PROGRAM Balanza_Semilla
VAR
	// grueso carga balanza
	TR_S_V2: Equipo_Valvula_5_2; //Válvula de corte grosso
	// fino carga balanza
	TR_S_V3: Equipo_Valvula_5_2;
	// descarga balanza
	TR_S_V4: Equipo_Valvula_5_2;
	//
	TR_S_V2_CmdAuto:BOOL;	//Válvula de corte grosso
	TR_S_V3_CmdAuto:BOOL;	//Válvula de corte fino
	TR_S_V4_CmdAuto:BOOL;	//Válvula de descarga
	// Balanza de pesaje de semilla
	TR_S_WT1: Balanza;
	//
	Hab_cargarSemilla	:BOOL;
	Cargar_Balanza		:BOOL;
	TolerInf_pesoSemilla:REAL;	//Tolerância inferior da carga da balança
	TolerSup_pesoSemilla:REAL;	//Tolerância superior da balança
	Balanza_cargadaOk	:BOOL;
	Hab_descargarSemilla:BOOL;
	Descargar_Balanza	:BOOL;
	PesoSemilla_paraDosificar:REAL;
	Espera_pesasArriba:TON;
	Espera_Estable:TON;
	Espera_DescAbierta:TON;
	
	// tiempo de carga/descarga de balanza semilla excesivo
	Alr_demoraCarga: TON;
	Alr_demoraDescarga:TON;
	
	TriggerTomarPeso :BOOL;
	
	//provisorios
	bHS :BOOL;
	dintHS	:DINT:=3;
	Hx :BOOL;
	IniCal:BOOL;
	
	iStep :INT;
	Espera_pesas :TON;
	
	AuxHugo :BOOL;
	Procesando: BOOL;
	Tabla_FIFO_Peso: Tabla_FIFO;
	Balanza_vacia: BOOL;
	FinCarga: BOOL;
	TmrGruesoOk: TON;
	TBalanzaVacia: TON;
	PolvosOk: BOOL;
	// Timer para aparecer a popup de peso fora de tolerância
	TON_PesoForaTolerancia: TON;
	TON_DemoraCarga: TON;
	// Se a caixa superior estiver sem nível de sementes, permite que a semente remanescente seja carregada na balança
	EsvaziarCaixa: BOOL;
	qtdBateladas	:UDINT;	//Quantidade de bateladas feitas
END_VAR
VAR // added by the converter: edge detectors and wires of the graphical bodies
    _rt1, _rt2, _rt3, _rt4, _rt5, _rt6 : R_TRIG;
    _w1, _w2, _w3, _w4, _w5, _w6, _w7, _w8, _w9, _w10, _w11, _w12, _w13, _w14, _w15 : BOOL;
    _ft1 : F_TRIG;
END_VAR

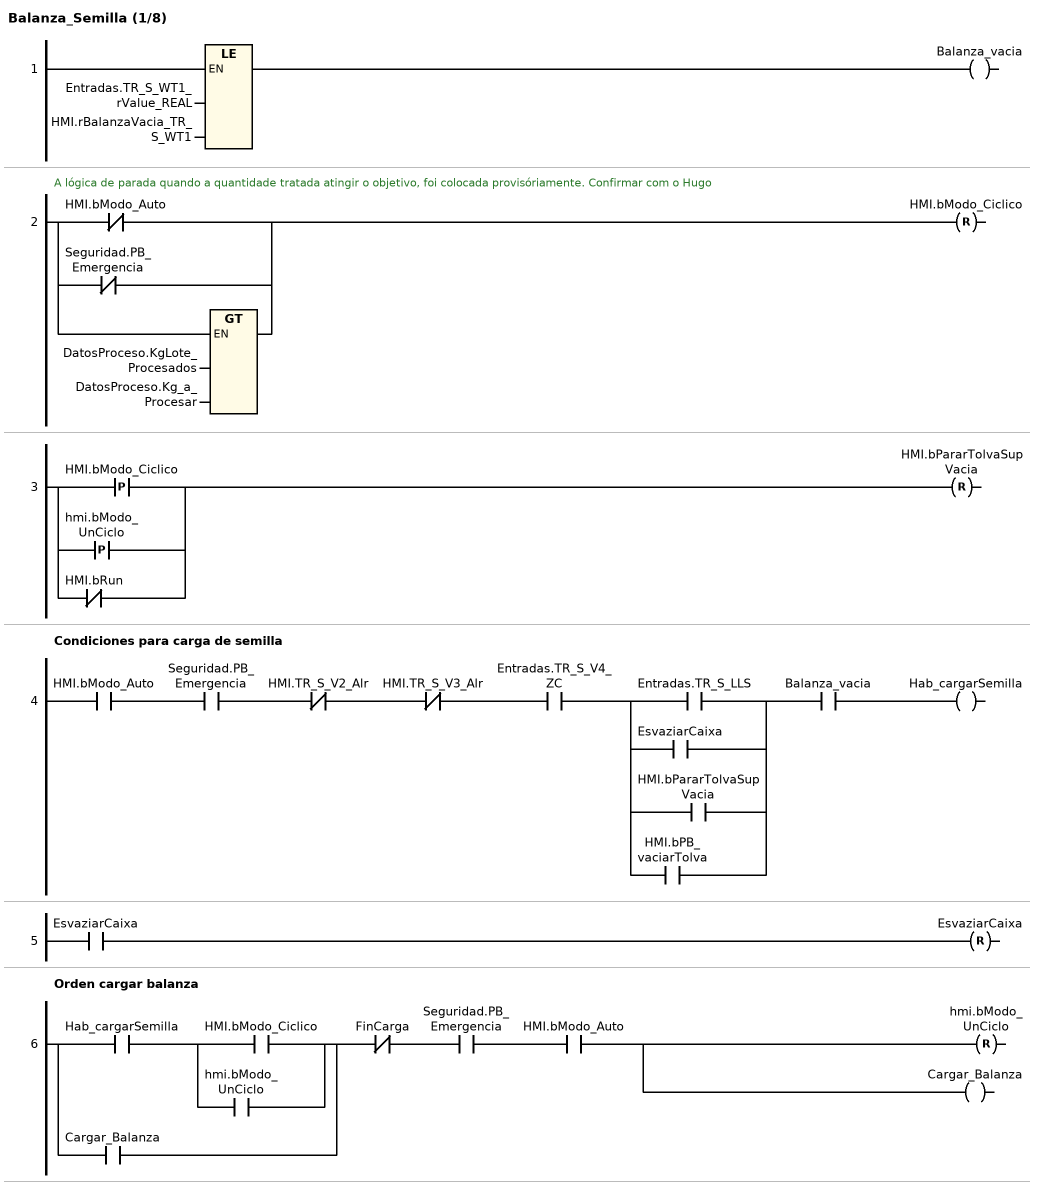
// NETWORK 1
Balanza_vacia := Entradas.TR_S_WT1_rValue_REAL <= HMI.rBalanzaVacia_TR_S_WT1;

// NETWORK 2
// A lógica de parada quando a quantidade tratada atingir o objetivo, foi colocada provisóriamente. Confirmar com o Hugo
HMI.bModo_Ciclico R= NOT HMI.bModo_Auto OR NOT Seguridad.PB_Emergencia OR DatosProceso.KgLote_Procesados > DatosProceso.Kg_a_Procesar;

// NETWORK 3
_rt1(CLK := HMI.bModo_Ciclico);
_rt2(CLK := hmi.bModo_UnCiclo);
HMI.bPararTolvaSupVacia R= _rt1.Q OR _rt2.Q OR NOT HMI.bRun;

// NETWORK 4: Condiciones para carga de semilla
Hab_cargarSemilla := HMI.bModo_Auto AND Seguridad.PB_Emergencia AND NOT HMI.TR_S_V2_Alr AND NOT HMI.TR_S_V3_Alr AND Entradas.TR_S_V4_ZC AND (Entradas.TR_S_LLS OR EsvaziarCaixa OR HMI.bPararTolvaSupVacia OR HMI.bPB_vaciarTolva) AND Balanza_vacia;

// NETWORK 5
EsvaziarCaixa R= EsvaziarCaixa;

// NETWORK 6: Orden cargar balanza
_w1 := (Hab_cargarSemilla AND (HMI.bModo_Ciclico OR hmi.bModo_UnCiclo) OR Cargar_Balanza) AND NOT FinCarga AND Seguridad.PB_Emergencia AND HMI.bModo_Auto;
hmi.bModo_UnCiclo R= _w1;
Cargar_Balanza := _w1;

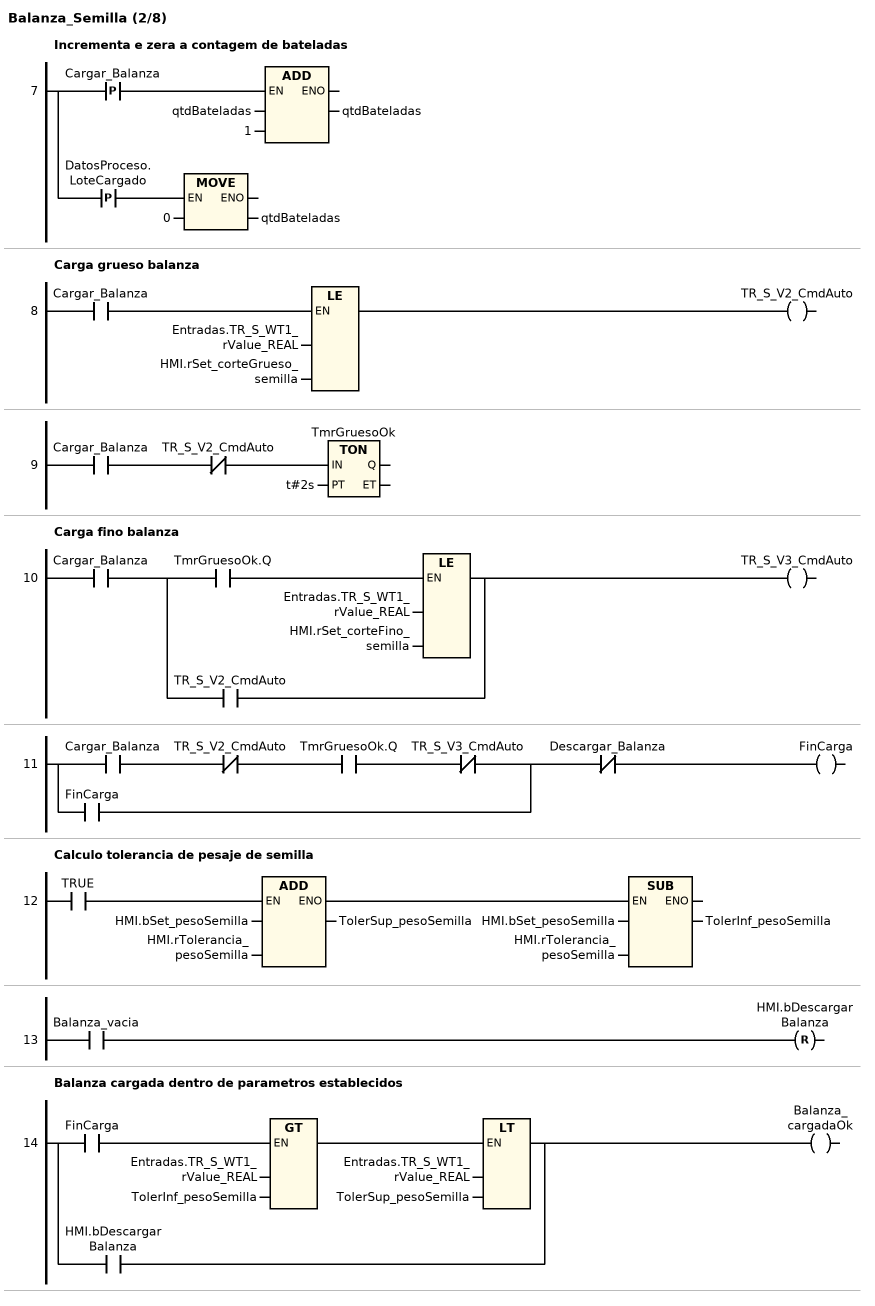
// NETWORK 7: Incrementa e zera a contagem de bateladas
_rt3(CLK := Cargar_Balanza);
_w2 := _rt3.Q;
IF _w2 THEN qtdBateladas := qtdBateladas + 1; END_IF
_rt4(CLK := DatosProceso.LoteCargado);
_w3 := _rt4.Q;
IF _w3 THEN qtdBateladas := 0; END_IF
(* _w2 OR _w3; result not used *)

// NETWORK 8: Carga grueso balanza
TR_S_V2_CmdAuto := Cargar_Balanza AND Entradas.TR_S_WT1_rValue_REAL <= HMI.rSet_corteGrueso_semilla;

// NETWORK 9
TmrGruesoOk(IN := Cargar_Balanza AND NOT TR_S_V2_CmdAuto, PT := t#2s); // TON

// NETWORK 10: Carga fino balanza
_w4 := Cargar_Balanza AND TR_S_V2_CmdAuto;
IF NOT _w4 THEN
    _w4 := Cargar_Balanza AND TmrGruesoOk.Q AND Entradas.TR_S_WT1_rValue_REAL <= HMI.rSet_corteFino_semilla;
END_IF
TR_S_V3_CmdAuto := _w4;

// NETWORK 11
FinCarga := (Cargar_Balanza AND NOT TR_S_V2_CmdAuto AND TmrGruesoOk.Q AND NOT TR_S_V3_CmdAuto OR FinCarga) AND NOT Descargar_Balanza;

// NETWORK 12: Calculo tolerancia de pesaje de semilla
TolerSup_pesoSemilla := HMI.bSet_pesoSemilla + HMI.rTolerancia_pesoSemilla;
TolerInf_pesoSemilla := HMI.bSet_pesoSemilla - HMI.rTolerancia_pesoSemilla;

// NETWORK 13
HMI.bDescargarBalanza R= Balanza_vacia;

// NETWORK 14: Balanza cargada dentro de parametros establecidos
_w5 := HMI.bDescargarBalanza;
IF NOT _w5 THEN
    _w5 := FinCarga AND Entradas.TR_S_WT1_rValue_REAL > TolerInf_pesoSemilla AND Entradas.TR_S_WT1_rValue_REAL < TolerSup_pesoSemilla;
END_IF
Balanza_cargadaOk := _w5;

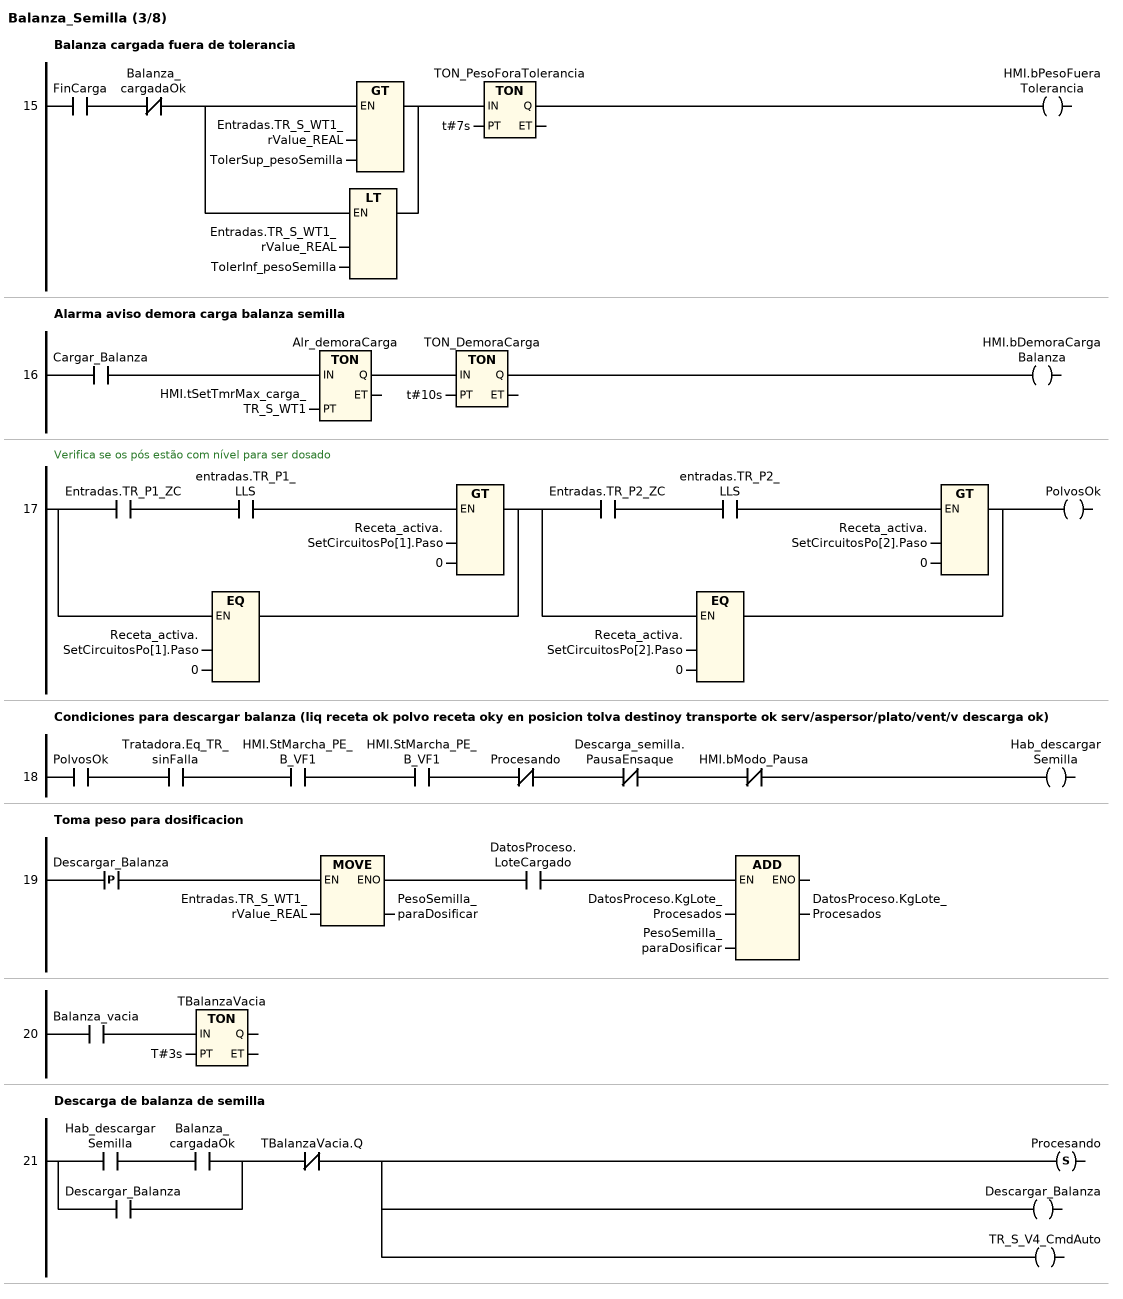
// NETWORK 15: Balanza cargada fuera de tolerancia
_w6 := FinCarga AND NOT Balanza_cargadaOk;
TON_PesoForaTolerancia(IN := _w6 AND Entradas.TR_S_WT1_rValue_REAL > TolerSup_pesoSemilla OR _w6 AND Entradas.TR_S_WT1_rValue_REAL < TolerInf_pesoSemilla, PT := t#7s); // TON
HMI.bPesoFueraTolerancia := TON_PesoForaTolerancia.Q;

// NETWORK 16: Alarma aviso demora carga balanza semilla
Alr_demoraCarga(IN := Cargar_Balanza, PT := HMI.tSetTmrMax_carga_TR_S_WT1); // TON
TON_DemoraCarga(IN := Alr_demoraCarga.Q, PT := t#10s); // TON
HMI.bDemoraCargaBalanza := TON_DemoraCarga.Q;

// NETWORK 17
// Verifica se os pós estão com nível para ser dosado
_w7 := Entradas.TR_P1_ZC AND entradas.TR_P1_LLS AND Receta_activa.SetCircuitosPo[1].Paso > 0 OR Receta_activa.SetCircuitosPo[1].Paso = 0;
PolvosOk := (_w7 AND Entradas.TR_P2_ZC) AND entradas.TR_P2_LLS AND Receta_activa.SetCircuitosPo[2].Paso > 0 OR _w7 AND Receta_activa.SetCircuitosPo[2].Paso = 0;

// NETWORK 18: Condiciones para descargar balanza (liq receta ok polvo receta oky en posicion tolva destinoy transporte ok serv/aspersor/plato/vent/v descarga ok)
Hab_descargarSemilla := PolvosOk AND Tratadora.Eq_TR_sinFalla AND HMI.StMarcha_PE_B_VF1 AND HMI.StMarcha_PE_B_VF1 AND NOT Procesando AND NOT Descarga_semilla.PausaEnsaque AND NOT HMI.bModo_Pausa;

// NETWORK 19: Toma peso para dosificacion
_rt5(CLK := Descargar_Balanza);
_w8 := _rt5.Q;
IF _w8 THEN PesoSemilla_paraDosificar := Entradas.TR_S_WT1_rValue_REAL; END_IF
IF _w8 AND DatosProceso.LoteCargado THEN
    DatosProceso.KgLote_Procesados := DatosProceso.KgLote_Procesados + PesoSemilla_paraDosificar;
END_IF

// NETWORK 20
TBalanzaVacia(IN := Balanza_vacia, PT := T#3s); // TON

// NETWORK 21: Descarga de balanza de semilla
_w9 := (Hab_descargarSemilla AND Balanza_cargadaOk OR Descargar_Balanza) AND NOT TBalanzaVacia.Q;
Procesando S= _w9;
Descargar_Balanza := _w9;
TR_S_V4_CmdAuto := _w9;

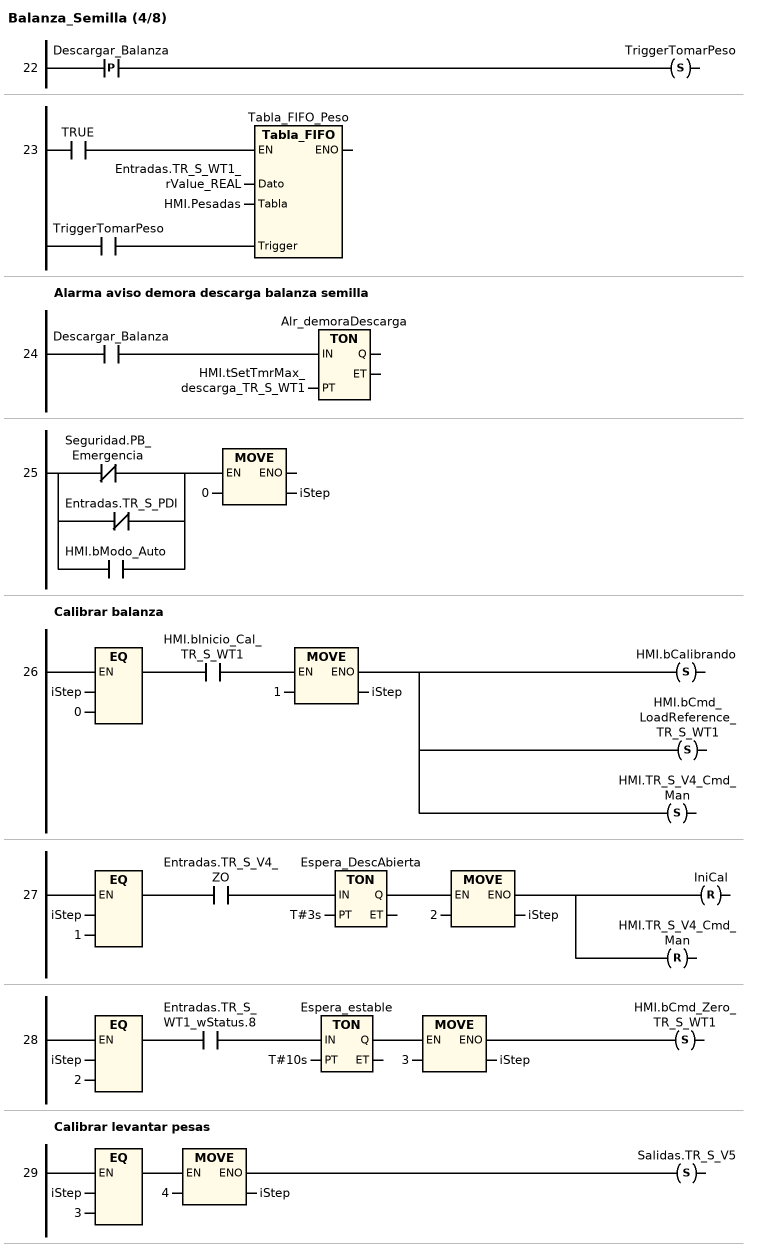
// NETWORK 22
_rt6(CLK := Descargar_Balanza);
TriggerTomarPeso S= _rt6.Q;

// NETWORK 23
Tabla_FIFO_Peso(Dato := Entradas.TR_S_WT1_rValue_REAL, Tabla := HMI.Pesadas, Trigger := TriggerTomarPeso); // Tabla_FIFO

// NETWORK 24: Alarma aviso demora descarga balanza semilla
Alr_demoraDescarga(IN := Descargar_Balanza, PT := HMI.tSetTmrMax_descarga_TR_S_WT1); // TON

// NETWORK 25
IF NOT Seguridad.PB_Emergencia OR NOT Entradas.TR_S_PDI OR HMI.bModo_Auto THEN iStep := 0; END_IF

// NETWORK 26: Calibrar balanza
_w10 := iStep = 0 AND HMI.bInicio_Cal_TR_S_WT1;
IF _w10 THEN iStep := 1; END_IF
HMI.bCalibrando S= _w10;
HMI.bCmd_LoadReference_TR_S_WT1 S= _w10;
HMI.TR_S_V4_Cmd_Man S= _w10;

// NETWORK 27
Espera_DescAbierta(IN := iStep = 1 AND Entradas.TR_S_V4_ZO, PT := T#3s); // TON
_w11 := Espera_DescAbierta.Q;
IF _w11 THEN iStep := 2; END_IF
IniCal R= _w11;
HMI.TR_S_V4_Cmd_Man R= _w11;

// NETWORK 28
Espera_estable(IN := iStep = 2 AND Entradas.TR_S_WT1_wStatus.8, PT := T#10s); // TON
_w12 := Espera_estable.Q;
IF _w12 THEN iStep := 3; END_IF
HMI.bCmd_Zero_TR_S_WT1 S= _w12;

// NETWORK 29: Calibrar levantar pesas
_w13 := iStep = 3;
IF _w13 THEN iStep := 4; END_IF
Salidas.TR_S_V5 S= _w13;

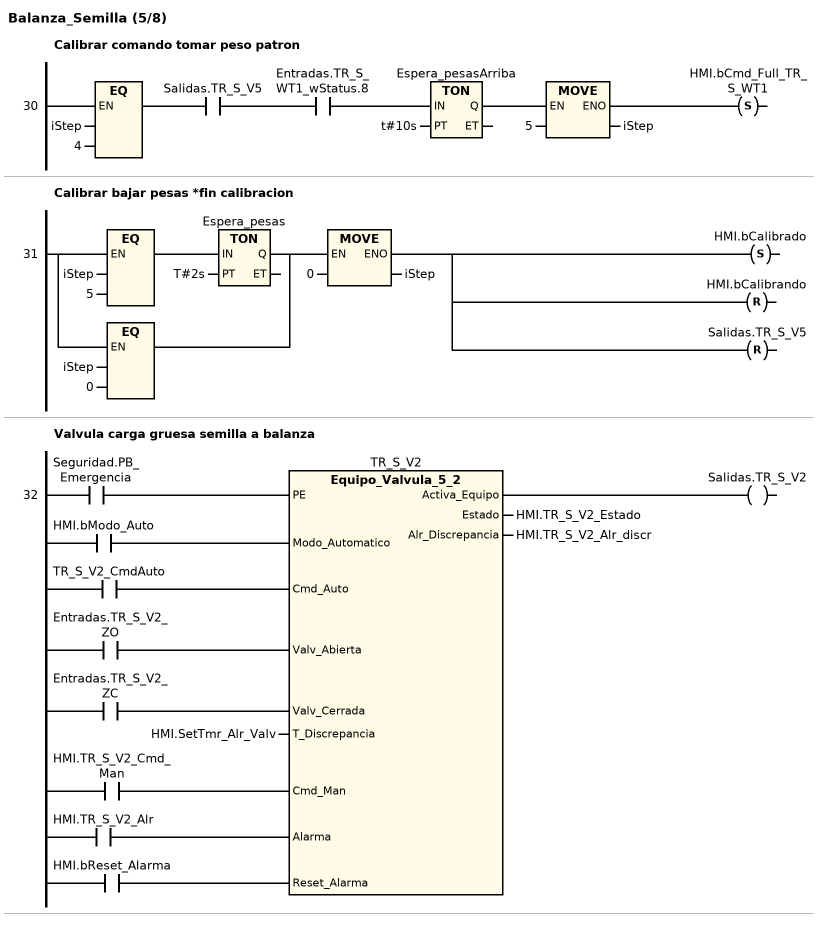
// NETWORK 30: Calibrar comando tomar peso patron
Espera_pesasArriba(IN := iStep = 4 AND Salidas.TR_S_V5 AND Entradas.TR_S_WT1_wStatus.8, PT := t#10s); // TON
_w14 := Espera_pesasArriba.Q;
IF _w14 THEN iStep := 5; END_IF
HMI.bCmd_Full_TR_S_WT1 S= _w14;

// NETWORK 31: Calibrar bajar pesas *fin calibracion
Espera_pesas(IN := iStep = 5, PT := T#2s); // TON
_w15 := Espera_pesas.Q OR iStep = 0;
IF _w15 THEN iStep := 0; END_IF
HMI.bCalibrado S= _w15;
HMI.bCalibrando R= _w15;
Salidas.TR_S_V5 R= _w15;

// NETWORK 32: Valvula carga gruesa semilla a balanza
TR_S_V2(
    PE := Seguridad.PB_Emergencia,
    Modo_Automatico := HMI.bModo_Auto,
    Cmd_Auto := TR_S_V2_CmdAuto,
    Valv_Abierta := Entradas.TR_S_V2_ZO,
    Valv_Cerrada := Entradas.TR_S_V2_ZC,
    T_Discrepancia := HMI.SetTmr_Alr_Valv,
    Cmd_Man := HMI.TR_S_V2_Cmd_Man,
    Alarma := HMI.TR_S_V2_Alr,
    Reset_Alarma := HMI.bReset_Alarma,
    Estado => HMI.TR_S_V2_Estado,
    Alr_Discrepancia => HMI.TR_S_V2_Alr_discr); // Equipo_Valvula_5_2
Salidas.TR_S_V2 := TR_S_V2.Activa_Equipo;

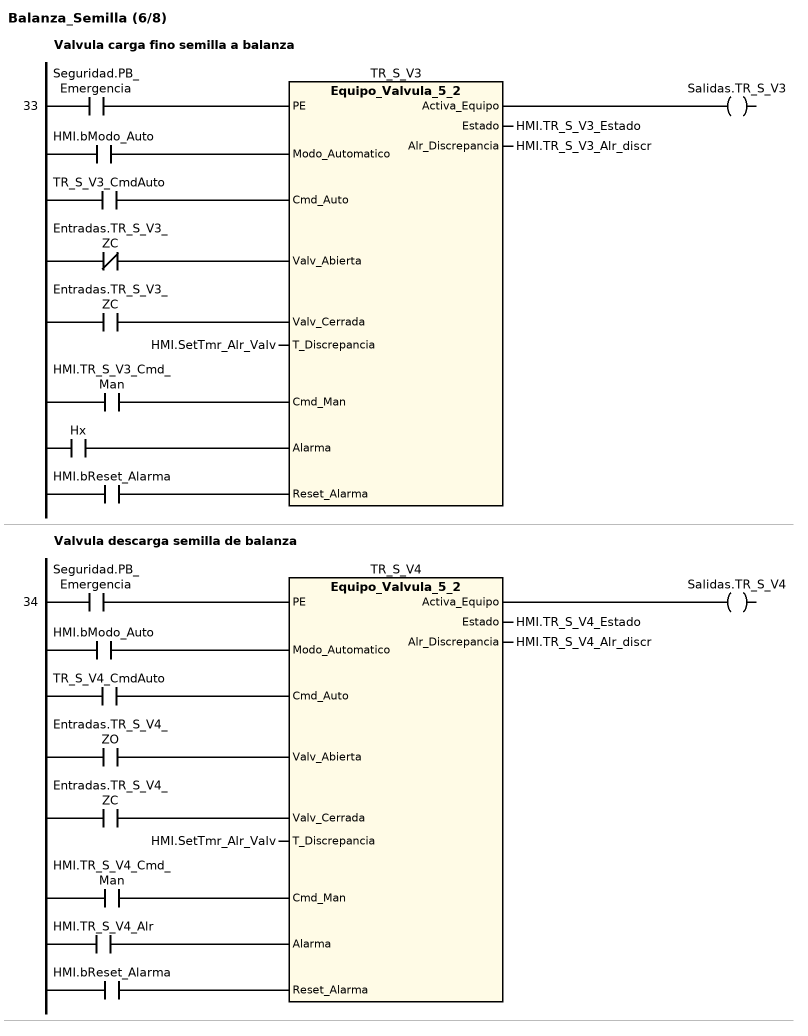
// NETWORK 33: Valvula carga fino semilla a balanza
TR_S_V3(
    PE := Seguridad.PB_Emergencia,
    Modo_Automatico := HMI.bModo_Auto,
    Cmd_Auto := TR_S_V3_CmdAuto,
    Valv_Abierta := NOT Entradas.TR_S_V3_ZC,
    Valv_Cerrada := Entradas.TR_S_V3_ZC,
    T_Discrepancia := HMI.SetTmr_Alr_Valv,
    Cmd_Man := HMI.TR_S_V3_Cmd_Man,
    Alarma := Hx,
    Reset_Alarma := HMI.bReset_Alarma,
    Estado => HMI.TR_S_V3_Estado,
    Alr_Discrepancia => HMI.TR_S_V3_Alr_discr); // Equipo_Valvula_5_2
Salidas.TR_S_V3 := TR_S_V3.Activa_Equipo;

// NETWORK 34: Valvula descarga semilla de balanza
TR_S_V4(
    PE := Seguridad.PB_Emergencia,
    Modo_Automatico := HMI.bModo_Auto,
    Cmd_Auto := TR_S_V4_CmdAuto,
    Valv_Abierta := Entradas.TR_S_V4_ZO,
    Valv_Cerrada := Entradas.TR_S_V4_ZC,
    T_Discrepancia := HMI.SetTmr_Alr_Valv,
    Cmd_Man := HMI.TR_S_V4_Cmd_Man,
    Alarma := HMI.TR_S_V4_Alr,
    Reset_Alarma := HMI.bReset_Alarma,
    Estado => HMI.TR_S_V4_Estado,
    Alr_Discrepancia => HMI.TR_S_V4_Alr_discr); // Equipo_Valvula_5_2
Salidas.TR_S_V4 := TR_S_V4.Activa_Equipo;

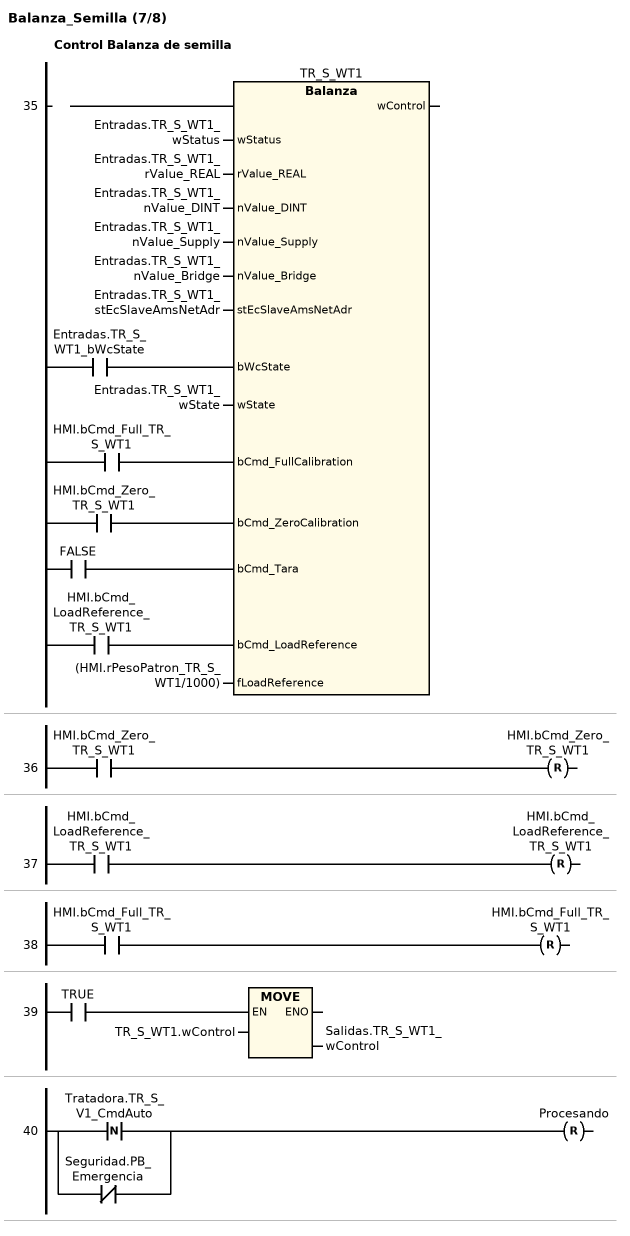
// NETWORK 35: Control Balanza de semilla
TR_S_WT1(
    wStatus := Entradas.TR_S_WT1_wStatus,
    rValue_REAL := Entradas.TR_S_WT1_rValue_REAL,
    nValue_DINT := Entradas.TR_S_WT1_nValue_DINT,
    nValue_Supply := Entradas.TR_S_WT1_nValue_Supply,
    nValue_Bridge := Entradas.TR_S_WT1_nValue_Bridge,
    stEcSlaveAmsNetAdr := Entradas.TR_S_WT1_stEcSlaveAmsNetAdr,
    bWcState := Entradas.TR_S_WT1_bWcState,
    wState := Entradas.TR_S_WT1_wState,
    bCmd_FullCalibration := HMI.bCmd_Full_TR_S_WT1,
    bCmd_ZeroCalibration := HMI.bCmd_Zero_TR_S_WT1,
    bCmd_Tara := FALSE,
    bCmd_LoadReference := HMI.bCmd_LoadReference_TR_S_WT1,
    fLoadReference := (HMI.rPesoPatron_TR_S_WT1/1000)); // Balanza

// NETWORK 36
HMI.bCmd_Zero_TR_S_WT1 R= HMI.bCmd_Zero_TR_S_WT1;

// NETWORK 37
HMI.bCmd_LoadReference_TR_S_WT1 R= HMI.bCmd_LoadReference_TR_S_WT1;

// NETWORK 38
HMI.bCmd_Full_TR_S_WT1 R= HMI.bCmd_Full_TR_S_WT1;

// NETWORK 39
Salidas.TR_S_WT1_wControl := TR_S_WT1.wControl;

// NETWORK 40
_ft1(CLK := Tratadora.TR_S_V1_CmdAuto);
Procesando R= _ft1.Q OR NOT Seguridad.PB_Emergencia;

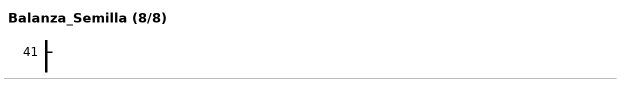
// NETWORK 41

END_PROGRAM

(* stored: Version 1.1.0.1, ProductVersion 3.1.4024.14
   POU Balanza_Semilla: Id {46f64667-312e-41a1-944c-3429d544bd42}, SpecialFunc None *)
